// TIA Portal V20 export
FUNCTION_BLOCK "SysMotor"   // FB2060, FBD
TITLE = manage a motor with contactor equipment
{ S7_Optimized_Access := 'TRUE' }
AUTHOR : MiCROTEC
VERSION : 1.6
// -2017.03 : Martin
// stored: AutoNumber false, MemoryReserve 100, SetENOAutomatically false
   VAR_INPUT
      area { ExternalAccessible := 'False'; ExternalVisible := 'False'; ExternalWritable := 'False'} : Bool;   // 1=safety area on
      auto { ExternalAccessible := 'False'; ExternalVisible := 'False'; ExternalWritable := 'False'} : Bool;   // automatic
      manP { ExternalAccessible := 'False'; ExternalVisible := 'False'; ExternalWritable := 'False'} : Bool;   // manual plus
      manM { ExternalAccessible := 'False'; ExternalVisible := 'False'; ExternalWritable := 'False'} : Bool;   // manual minus
      autoP { ExternalAccessible := 'False'; ExternalVisible := 'False'; ExternalWritable := 'False'} : Bool;   // automatic plus
      autoM { ExternalAccessible := 'False'; ExternalVisible := 'False'; ExternalWritable := 'False'} : Bool;   // automatic minus
      ack { ExternalAccessible := 'False'; ExternalVisible := 'False'; ExternalWritable := 'False'} : Bool;   // fault acknowledge
      lampTest { ExternalAccessible := 'False'; ExternalVisible := 'False'; ExternalWritable := 'False'} : Bool;   // lamptest
      enableP { ExternalAccessible := 'False'; ExternalVisible := 'False'; ExternalWritable := 'False'} : Bool;   // release plus
      enableM { ExternalAccessible := 'False'; ExternalVisible := 'False'; ExternalWritable := 'False'} : Bool;   // release minus
      enAutoP { ExternalAccessible := 'False'; ExternalVisible := 'False'; ExternalWritable := 'False'} : Bool;   // release automatic plus
      enAutoM { ExternalAccessible := 'False'; ExternalVisible := 'False'; ExternalWritable := 'False'} : Bool;   // release automatic minus
      mpMotor { ExternalAccessible := 'False'; ExternalVisible := 'False'; ExternalWritable := 'False'} : Bool;   // 1=motor protection switch ok
      mpBrake { ExternalAccessible := 'False'; ExternalVisible := 'False'; ExternalWritable := 'False'} : Bool;   // 1=motor protection switch brake ok
      mpBrake2 { ExternalAccessible := 'False'; ExternalVisible := 'False'; ExternalWritable := 'False'} : Bool;   // 1=motor protection switch brake ok
      mpFan { ExternalAccessible := 'False'; ExternalVisible := 'False'; ExternalWritable := 'False'} : Bool;   // 1=motor protection switch fan ok
      thMotor { ExternalAccessible := 'False'; ExternalVisible := 'False'; ExternalWritable := 'False'} : Bool;   // 1=thermal contact motor ok
      thMotorRtd { ExternalAccessible := 'False'; ExternalVisible := 'False'; ExternalWritable := 'False'} : Int;   // thermal contact motor AE 8xRTD
      mSwitch { ExternalAccessible := 'False'; ExternalVisible := 'False'; ExternalWritable := 'False'} : Bool;   // 1=maintenance switch is ok
      fdb { ExternalAccessible := 'False'; ExternalVisible := 'False'; ExternalWritable := 'False'} : Bool;   // 1=feedback circuit ok
      changeDirTime { ExternalAccessible := 'False'; ExternalVisible := 'False'; ExternalWritable := 'False'} : Time := T#500MS;   // time wait to restart in oder direction
      restartTime { ExternalAccessible := 'False'; ExternalVisible := 'False'; ExternalWritable := 'False'} : Time := T#500MS;   // time wait to restart in any direction
      brakeOnTime { ExternalAccessible := 'False'; ExternalVisible := 'False'; ExternalWritable := 'False'} : Time := T#10MS;   // time wait to open the brake
      brakeOffTime { ExternalAccessible := 'False'; ExternalVisible := 'False'; ExternalWritable := 'False'} : Time := T#10MS;   // time wait to close the brake
      metPerMin { ExternalAccessible := 'False'; ExternalVisible := 'False'; ExternalWritable := 'False'} : Real := 1.0;   // meter per minute with nominal speed
      cycle { ExternalAccessible := 'False'; ExternalVisible := 'False'; ExternalWritable := 'False'} : Real;   // cycle
   END_VAR
   VAR_OUTPUT
      plus { ExternalAccessible := 'False'; ExternalVisible := 'False'; ExternalWritable := 'False'} : Bool;   // drive plus
      minus { ExternalAccessible := 'False'; ExternalVisible := 'False'; ExternalWritable := 'False'} : Bool;   // drive minus
      brake { ExternalAccessible := 'False'; ExternalVisible := 'False'; ExternalWritable := 'False'} : Bool;   // brake open
      brake2 { ExternalAccessible := 'False'; ExternalVisible := 'False'; ExternalWritable := 'False'} : Bool;   // brake open
      enStartP { ExternalAccessible := 'False'; ExternalVisible := 'False'; ExternalWritable := 'False'} : Bool;   // release drive plus
      enStartM { ExternalAccessible := 'False'; ExternalVisible := 'False'; ExternalWritable := 'False'} : Bool;   // release drive minus
      fan { ExternalAccessible := 'False'; ExternalVisible := 'False'; ExternalWritable := 'False'} : Bool;   // fan on
      lamp { ExternalAccessible := 'False'; ExternalVisible := 'False'; ExternalWritable := 'False'} : Bool;   // indication lamp
      lamp2 { ExternalAccessible := 'False'; ExternalVisible := 'False'; ExternalWritable := 'False'} : Bool;   // indication lamp 2
      actSpeed { ExternalAccessible := 'False'; ExternalVisible := 'False'; ExternalWritable := 'False'} : Real;   // actual speed
      mmCycle { ExternalAccessible := 'False'; ExternalVisible := 'False'; ExternalWritable := 'False'} : Real;   // milimeter per cycle
      err { ExternalAccessible := 'False'; ExternalVisible := 'False'; ExternalWritable := 'False'} : Bool;   // fault
   END_VAR
   VAR_IN_OUT
      Mot : "TypeMotor";   // Daten an VISU Motor
   END_VAR
   VAR
      var { ExternalAccessible := 'False'; ExternalVisible := 'False'; ExternalWritable := 'False'} : Struct
         true : Bool;
         false : Bool;
         "bool" : Bool;
         "byte" : Byte;
         "word" : Word;
         "dword" : DWord;
         "int" : Int;
         "dint" : DInt;
         "real" : Real;
         s5time : S5Time;
         "time" : Time;
         hm : Array[1..50] of Bool;
         fm : Array[1..50] of Bool;
      END_STRUCT;
      T { ExternalAccessible := 'False'; ExternalVisible := 'False'; ExternalWritable := 'False'} : Array[1..15] of IEC_TIMER;
      restartBreak { ExternalAccessible := 'False'; ExternalVisible := 'False'; ExternalWritable := 'False'} : Bool;
      man { ExternalAccessible := 'False'; ExternalVisible := 'False'; ExternalWritable := 'False'} : Bool;
      changeDirDelM { ExternalAccessible := 'False'; ExternalVisible := 'False'; ExternalWritable := 'False'} : Bool;
      changeDirDelP { ExternalAccessible := 'False'; ExternalVisible := 'False'; ExternalWritable := 'False'} : Bool;
      mpFanOffDel { ExternalAccessible := 'False'; ExternalVisible := 'False'; ExternalWritable := 'False'} : Bool;
      brakeOnDel { ExternalAccessible := 'False'; ExternalVisible := 'False'; ExternalWritable := 'False'} : Bool;
      brakeOffDel { ExternalAccessible := 'False'; ExternalVisible := 'False'; ExternalWritable := 'False'} : Bool;
      autoOld { ExternalAccessible := 'False'; ExternalVisible := 'False'; ExternalWritable := 'False'} : Bool;
   END_VAR
   VAR_TEMP
      tempAck : Bool;
   END_VAR
   VAR_TEMP   // added for the SCL form of the ladder/FBD networks
      _w1 : Bool;
      _w2 : Bool;
   END_VAR
BEGIN

REGION Network 1: ack
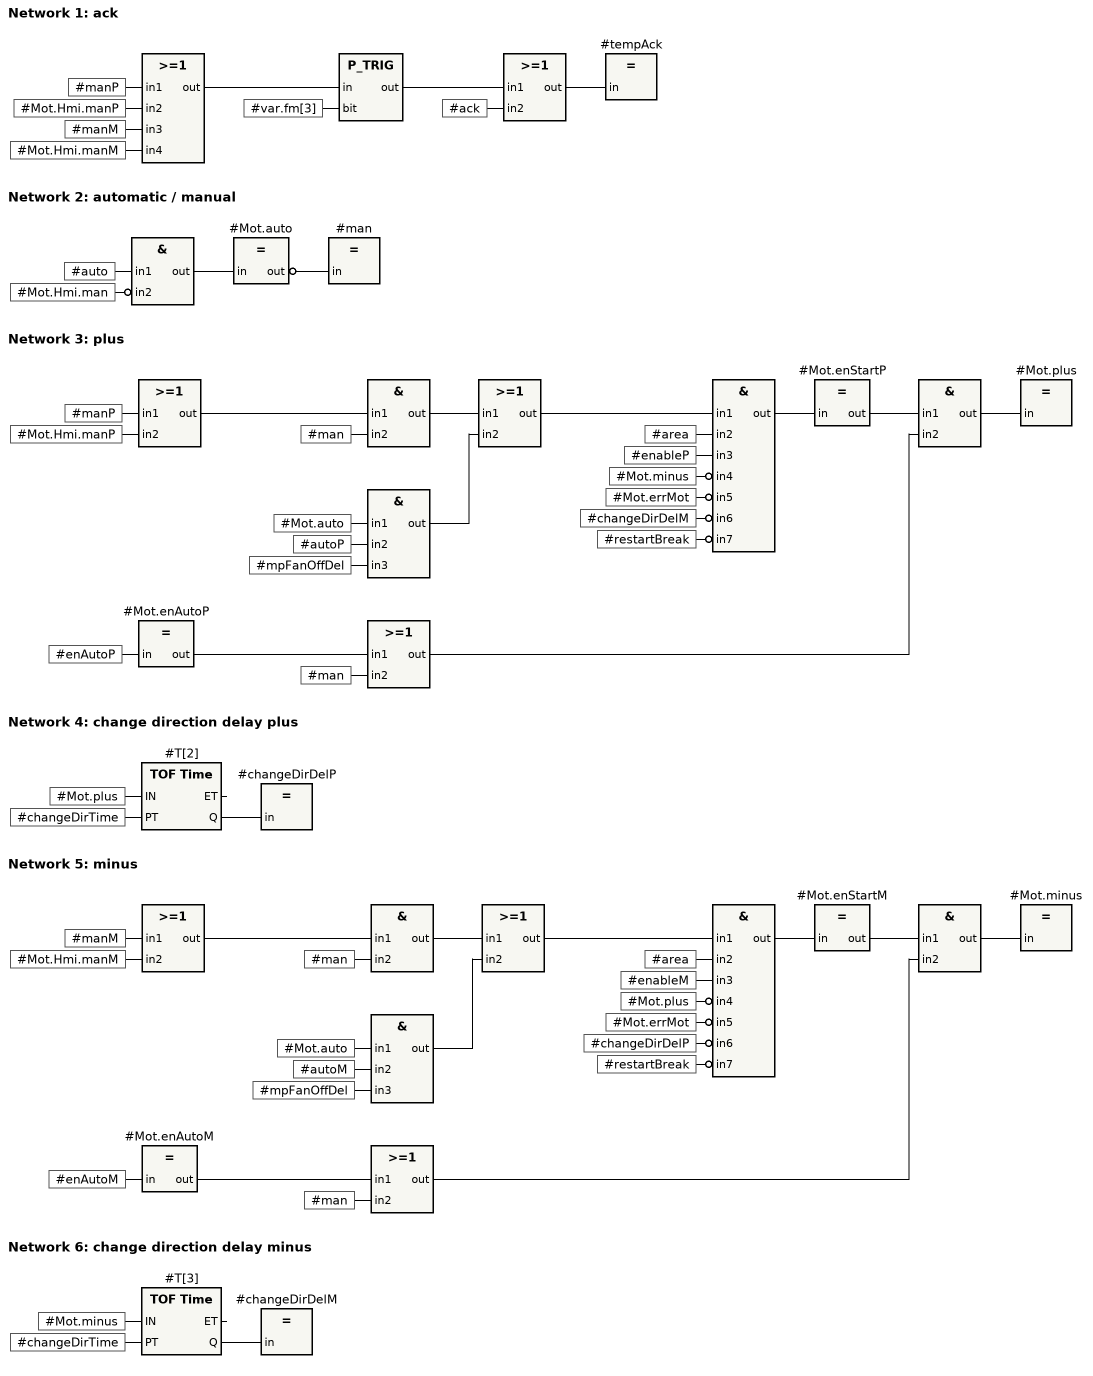
   #_w1 := #manP OR #Mot.Hmi.manP OR #manM OR #Mot.Hmi.manM;
   #_w2 := #_w1 AND NOT #var.fm[3];   // rising edge
   #var.fm[3] := #_w1;
   #tempAck := #_w2 OR #ack;
END_REGION

REGION Network 2: automatic / manual
   #_w1 := #auto AND NOT #Mot.Hmi.man;
   #Mot.auto := #_w1;
   #man := NOT #_w1;
END_REGION

REGION Network 3: plus
   #Mot.enStartP := (((#manP OR #Mot.Hmi.manP) AND #man) OR (#Mot.auto AND #autoP AND #mpFanOffDel)) AND #area AND #enableP AND NOT #Mot.minus AND NOT #Mot.errMot AND NOT #changeDirDelM AND NOT #restartBreak;
   #Mot.enAutoP := #enAutoP;
   #Mot.plus := #Mot.enStartP AND (#enAutoP OR #man);
END_REGION

REGION Network 4: change direction delay plus
   #T[2].TOF(IN := #Mot.plus, PT := #changeDirTime);
   #changeDirDelP := #T[2].Q;
END_REGION

REGION Network 5: minus
   #Mot.enStartM := (((#manM OR #Mot.Hmi.manM) AND #man) OR (#Mot.auto AND #autoM AND #mpFanOffDel)) AND #area AND #enableM AND NOT #Mot.plus AND NOT #Mot.errMot AND NOT #changeDirDelP AND NOT #restartBreak;
   #Mot.enAutoM := #enAutoM;
   #Mot.minus := #Mot.enStartM AND (#enAutoM OR #man);
END_REGION

REGION Network 6: change direction delay minus
   #T[3].TOF(IN := #Mot.minus, PT := #changeDirTime);
   #changeDirDelM := #T[3].Q;
END_REGION

REGION Network 7: restart delay
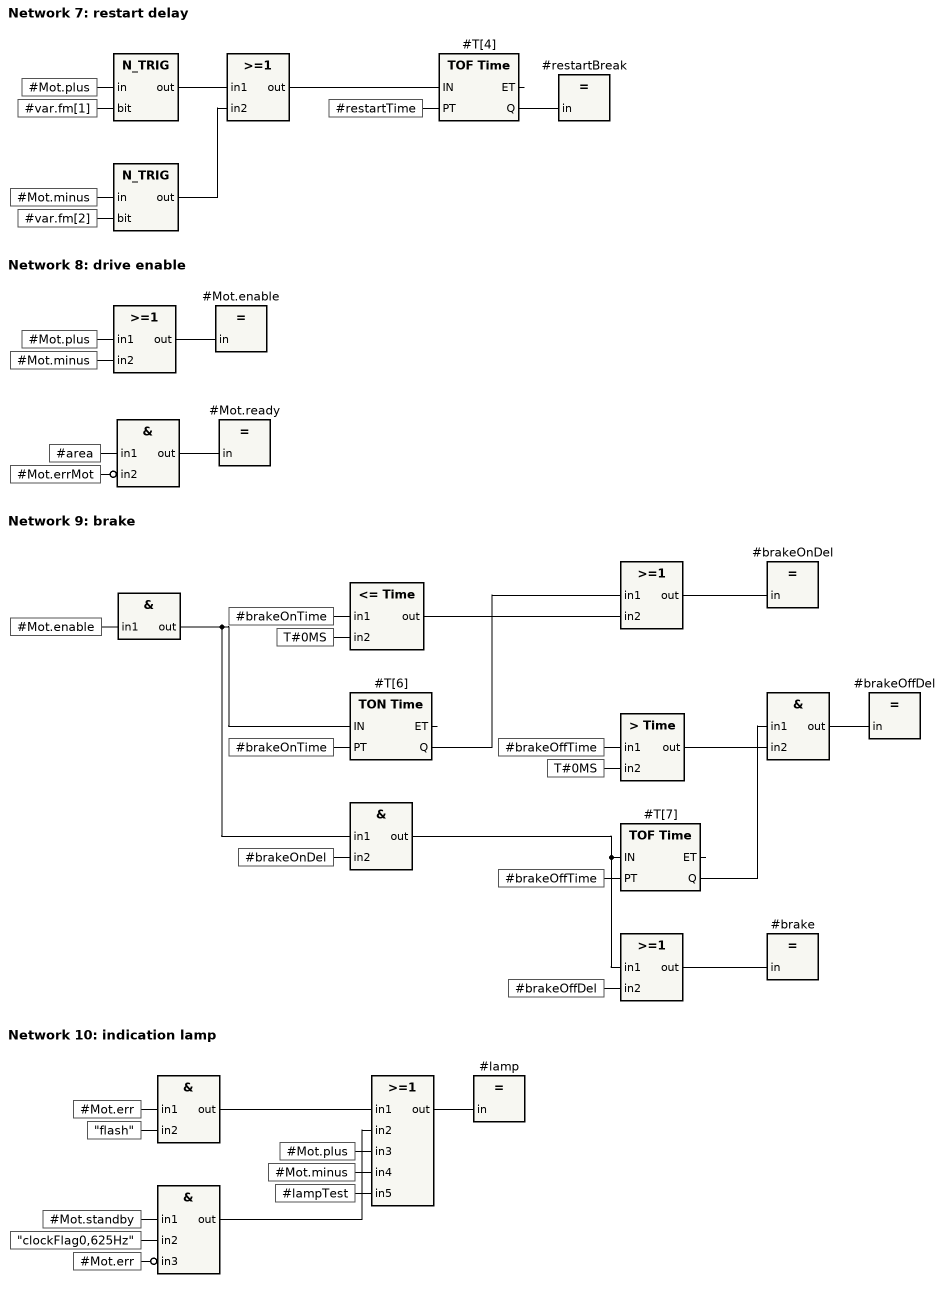
   #_w1 := NOT #Mot.plus AND #var.fm[1];   // falling edge
   #var.fm[1] := #Mot.plus;
   #_w2 := NOT #Mot.minus AND #var.fm[2];   // falling edge
   #var.fm[2] := #Mot.minus;
   #T[4].TOF(IN := #_w1 OR #_w2, PT := #restartTime);
   #restartBreak := #T[4].Q;
END_REGION

REGION Network 8: drive enable
   #Mot.enable := #Mot.plus OR #Mot.minus;
   #Mot.ready := #area AND NOT #Mot.errMot;
END_REGION

REGION Network 9: brake
   #T[6].TON(IN := #Mot.enable, PT := #brakeOnTime);
   #brakeOnDel := #T[6].Q OR (#brakeOnTime <= T#0MS);
   #_w1 := #Mot.enable AND #brakeOnDel;
   #T[7].TOF(IN := #_w1, PT := #brakeOffTime);
   #brakeOffDel := #T[7].Q AND (#brakeOffTime > T#0MS);
   #brake := #_w1 OR #brakeOffDel;
END_REGION

REGION Network 10: indication lamp
   #lamp := (#Mot.err AND "flash") OR (#Mot.standby AND "clockFlag0,625Hz" AND NOT #Mot.err) OR #Mot.plus OR #Mot.minus OR #lampTest;
END_REGION

REGION Network 11: direction plus delayed
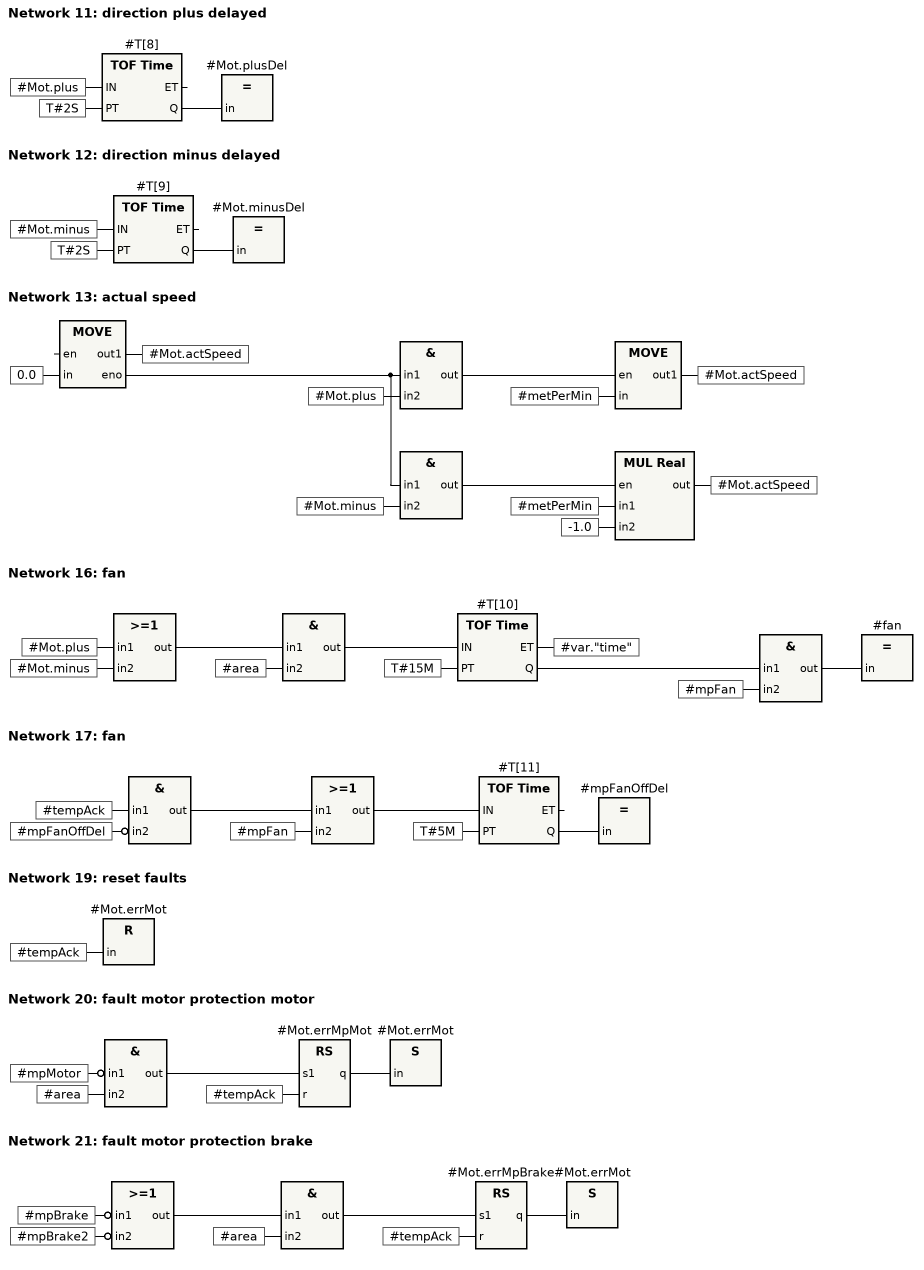
   #T[8].TOF(IN := #Mot.plus, PT := T#2S);
   #Mot.plusDel := #T[8].Q;
END_REGION

REGION Network 12: direction minus delayed
   #T[9].TOF(IN := #Mot.minus, PT := T#2S);
   #Mot.minusDel := #T[9].Q;
END_REGION

REGION Network 13: actual speed
   // ENO of a box is taken as its EN; it also drops when the box reports an error
   #Mot.actSpeed := 0.0;
   IF #Mot.plus THEN #Mot.actSpeed := #metPerMin; END_IF;
   IF #Mot.minus THEN #Mot.actSpeed := #metPerMin * (-1.0); END_IF;
END_REGION

REGION Network 14 (SCL): millimeter per cycle
   #Mot.mmCycle := 0.0;
   IF #Mot.plus OR #Mot.minus THEN
      #Mot.mmCycle := (#cycle *  #Mot.actSpeed ) / 60.0;
   END_IF;
END_REGION

REGION Network 15: -- fan--
END_REGION

REGION Network 16: fan
   #T[10].TOF(IN := (#Mot.plus OR #Mot.minus) AND #area, PT := T#15M, ET => #var."time");
   #fan := #T[10].Q AND #mpFan;
END_REGION

REGION Network 17: fan
   #T[11].TOF(IN := (#tempAck AND NOT #mpFanOffDel) OR #mpFan, PT := T#5M);
   #mpFanOffDel := #T[11].Q;
END_REGION

REGION Network 18: --faults--
END_REGION

REGION Network 19: reset faults
   IF #tempAck THEN #Mot.errMot := FALSE; END_IF;
END_REGION

REGION Network 20: fault motor protection motor
   IF #tempAck THEN
       #Mot.errMpMot := FALSE;   // RS flip-flop
   END_IF;
   IF NOT #mpMotor AND #area THEN #Mot.errMpMot := TRUE; END_IF;
   IF #Mot.errMpMot THEN #Mot.errMot := TRUE; END_IF;
END_REGION

REGION Network 21: fault motor protection brake
   IF #tempAck THEN
       #Mot.errMpBrake := FALSE;   // RS flip-flop
   END_IF;
   IF (NOT #mpBrake OR NOT #mpBrake2) AND #area THEN #Mot.errMpBrake := TRUE; END_IF;
   IF #Mot.errMpBrake THEN #Mot.errMot := TRUE; END_IF;
END_REGION

REGION Network 22: fault thermal contact motor
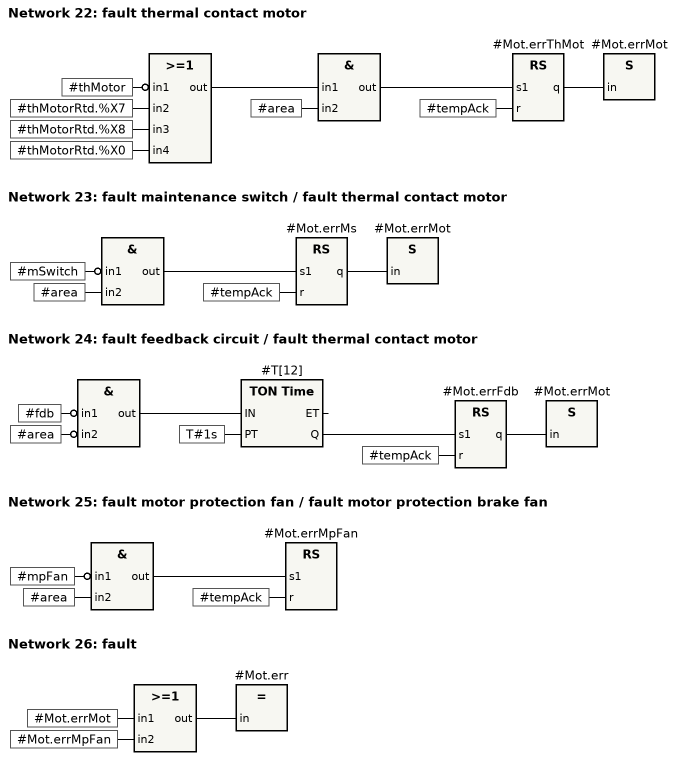
   IF #tempAck THEN
       #Mot.errThMot := FALSE;   // RS flip-flop
   END_IF;
   IF (NOT #thMotor OR #thMotorRtd.%X7 OR #thMotorRtd.%X8 OR #thMotorRtd.%X0) AND #area THEN
       #Mot.errThMot := TRUE;
   END_IF;
   IF #Mot.errThMot THEN #Mot.errMot := TRUE; END_IF;
END_REGION

REGION Network 23: fault maintenance switch / fault thermal contact motor
   IF #tempAck THEN
       #Mot.errMs := FALSE;   // RS flip-flop
   END_IF;
   IF NOT #mSwitch AND #area THEN #Mot.errMs := TRUE; END_IF;
   IF #Mot.errMs THEN #Mot.errMot := TRUE; END_IF;
END_REGION

REGION Network 24: fault feedback circuit / fault thermal contact motor
   #T[12].TON(IN := NOT #fdb AND NOT #area, PT := T#1s);
   IF #tempAck THEN
       #Mot.errFdb := FALSE;   // RS flip-flop
   END_IF;
   IF #T[12].Q THEN #Mot.errFdb := TRUE; END_IF;
   IF #Mot.errFdb THEN #Mot.errMot := TRUE; END_IF;
END_REGION

REGION Network 25: fault motor protection fan / fault motor protection brake fan
   IF #tempAck THEN
       #Mot.errMpFan := FALSE;   // RS flip-flop
   END_IF;
   IF NOT #mpFan AND #area THEN #Mot.errMpFan := TRUE; END_IF;
END_REGION

REGION Network 26: fault
   #Mot.err := #Mot.errMot OR #Mot.errMpFan;
END_REGION

REGION Network 27 (SCL): write outputs
      #plus := #Mot.plus;
      #minus := #Mot.minus;
      #brake2 := #brake;
      #enStartP :=  #Mot.enStartP ;
      #enStartM :=  #Mot.enStartM;
      #lamp2 :=#lamp;
      #err :=  #Mot.err;
      #actSpeed :=  #Mot.actSpeed ;
      #mmCycle := #Mot.mmCycle;
END_REGION

REGION Network 28 (SCL): in/out data
      #Mot.run := #Mot.plus OR #Mot.minus;
      #Mot.runDel :=  #Mot.plusDel  OR  #Mot.minusDel ;
      #Mot.errNr := 0;
      #Mot.tarSpeed := #metPerMin;
      #Mot.area := #area;

       IF #auto AND NOT #autoOld THEN
           #Mot.Hmi.man := false;
           #Mot.Hmi.manP := false;
           #Mot.Hmi.manM := false;
       END_IF;
       #autoOld := #auto;
END_REGION
END_FUNCTION_BLOCK
